// TIA Portal V16 export
// export: Created 2024-09-05T17:39:07.1020419Z, ExportSetting WithDefaults, DisplayName Totally Integrated Automation Portal, DisplayVersion V16 Update 6, DisplayName TIA Portal Version Control Interface, DisplayVersion V16 Update 2, DisplayName TIA Portal Openness, DisplayVersion V16 Update 6, DisplayName STEP 7 Professional, DisplayVersion V16 Update 6, DisplayName STEP 7 Safety, DisplayVersion V16, DisplayName WinCC Advanced, DisplayVersion V16 Update 6
DATA_BLOCK "AnalogData"   // DB27
{ S7_Optimized_Access := 'FALSE' }
VERSION : 0.1
// stored: AutoNumber false, DBAccessibleFromOPCUA true, IsOnlyStoredInLoadMemory false, IsWriteProtectedInAS false
   VAR
      InputResults : Array[1..12] of Real;
      OutputsRequired : Array[1..8] of Real;
      OutputsRequiredHMI : Array[1..8] of Int;
   END_VAR
BEGIN
   InputResults[1] := 7.960068;
   InputResults[2] := 8.440392;
   InputResults[3] := 7.105035;
   InputResults[4] := 7.011719;
   InputResults[5..12] := 0.0;
   OutputsRequired[1..8] := 0.0;
   OutputsRequiredHMI[1..8] := 16#0000;
END_DATA_BLOCK
